(* IEC 61131-3 sources: ABB_Hackathon/kb, 2 files *)

(* ---- alarm.st ---- *)
Title: Alarm Pattern (ST)

VAR
    PV : REAL; High : REAL; AlarmHigh : BOOL;
END_VAR

AlarmHigh := PV > High;
(* Add delay_on if needed with TON *)

(* ---- hysteresis.st ---- *)
Title: Hysteresis Control Template

VAR
    PV : REAL; (* Process value *)
    Cmd : BOOL; (* Output command *)
    High : REAL; Low : REAL; (* thresholds *)
END_VAR

IF (PV > High) THEN
    Cmd := TRUE;
ELSIF (PV < Low) THEN
    Cmd := FALSE;
END_IF;
